Fanuc KAREL source: NC0006.KL

-- PROVISIONAL review KL for V940-1; original PC SHA256 1065aa4dd0043d314ed55ce4366d893c015f7e90194a44f4d8804798a4b05649
-- Incomplete behavior may be omitted. Consult companion uncertainty JSON. Do not deploy.
PROGRAM NC0006
%NOLOCKGROUP
-- UNRESOLVED_LOCAL_POOL 1 cells at code offset 3; source declarations unknown
-- DIRECT_LOCAL_WORD_ACCESS alone does not prove INTEGER, REAL, or BOOLEAN
BEGIN
  -- V9_EXPOSED_INDEXED_TABLE_HINT layout=0001; 16 counted words exposed once; source arms/runtime held
  -- V9_CONDITION_STACK_HINT 8 bounded expression windows; static native code-base-relative target link; source arms held
  -- UNRESOLVED_PC offsets 0-8; opcodes 2B,2C,7B
  -- UNRESOLVED_PC offsets 13-20; opcodes 9D,23
  -- UNRESOLVED_PC offsets 25-38; opcodes 21,9D,57,79
  -- UNRESOLVED_PC offsets 43-56; opcodes 21,9D,57,79
  -- UNRESOLVED_PC offsets 61-74; opcodes 21,9D,57,79
  -- UNRESOLVED_PC offsets 79-92; opcodes 21,9D,57,79
  -- UNRESOLVED_PC offsets 97-110; opcodes 21,9D,57,79
  -- UNRESOLVED_PC offsets 115-128; opcodes 21,9D,57,79
  -- UNRESOLVED_PC offsets 133-146; opcodes 21,9D,57,79
  -- UNRESOLVED_PC offsets 151-164; opcodes 21,9D,57,79
  -- UNRESOLVED_PC offsets 169-183; opcodes 21,9D,52,23
  -- UNRESOLVED_PC offsets 188-193; opcodes 7A
  -- UNRESOLVED_PC offsets 198-216; opcodes 21,2E,52,23
  -- UNRESOLVED_PC offsets 226-231; opcodes 7A
  -- UNRESOLVED_PC offsets 236-254; opcodes 21,2E,52,23
  -- UNRESOLVED_PC offsets 264-269; opcodes 7A
  -- UNRESOLVED_PC offsets 274-292; opcodes 21,2E,52,23
  -- UNRESOLVED_PC offsets 302-307; opcodes 7A
  -- UNRESOLVED_PC offsets 312-330; opcodes 21,2E,52,23
  -- UNRESOLVED_PC offsets 340-345; opcodes 7A
  -- UNRESOLVED_PC offsets 350-368; opcodes 21,2E,52,23
  -- UNRESOLVED_PC offsets 378-383; opcodes 7A
  -- UNRESOLVED_PC offsets 388-406; opcodes 21,2E,52,23
  -- UNRESOLVED_PC offsets 416-421; opcodes 7A
  -- UNRESOLVED_PC offsets 426-444; opcodes 21,2E,52,23
  -- UNRESOLVED_PC offsets 454-459; opcodes 7A
  -- UNRESOLVED_PC offsets 464-482; opcodes 21,2E,52,23
  -- UNRESOLVED_PC offsets 492-496; opcodes 7F
  -- UNRESOLVED_PC offsets 501-505; opcodes 27,AA
  -- UNRESOLVED_PC offsets 510-514; opcodes 7F
END NC0006
